// TIA Portal V21 export
DATA_BLOCK "FB_Sensores_DB"   // DB2
// stored: InstanceOfName FB_Sensores, InstanceOfType FB
"FB_Sensores"
   // VAR_INPUT
   //    High_sensor : Bool;
   //    Low_sensor : Bool;
   //    "At left" : Bool;
   //    "At right" : Bool;
   //    Reset_estados : Bool;
   //    Loaded : Bool;
   //    "At left exit" : Bool;
   //    "At right exit" : Bool;
   // END_VAR
   // VAR_OUTPUT
   //    Clasificando : Bool;
   //    "Caja Alta" : Bool;
   //    "Caja Baja" : Bool;
   // END_VAR
   // VAR_IN_OUT
   //    CT_Total : Int;
   //    CT_Cajas_Altas : Int;
   //    CT_Cajas_Bajas : Int;
   // END_VAR
   // VAR
   //    Mem_At_left : Bool;
   //    Mem_At_right : Bool;
   //    Mem_clasificando : Bool;
   //    Mem_At_left_exit : Bool;
   //    Mem_At_right_exit : Bool;
   // END_VAR
BEGIN
END_DATA_BLOCK
